FUNCTION_BLOCK Test_AssertEquals_BOOL EXTENDS TUnitTestBase
VAR
    AssertionUnderTest : TAssertion(AssertionListenerMock);
    AssertionListenerMock : TAssertionListenerMock;
    BOOL_Variable : BOOL := FALSE;
END_VAR

AssertionListenerMock.AssertionFailed  := FALSE;
AssertionListenerMock.AssertionMessage := '';
AssertionListenerMock.ExpectedAsString := '';
AssertionListenerMock.ActualAsString   := '';

// Test the assertion...
AssertionUnderTest.AssertEquals_BOOL(
    Expected := TRUE,
    Actual   := BOOL_Variable,
    VariableName := 'BOOL_Variable');
    
// Check the assertion worked...    
Assertion.AssertEquals_BOOL(
    Expected := TRUE,
    Actual   := AssertionListenerMock.AssertionFailed,
    VariableName := 'AssertionListenerMock.AssertionFailed');

// Check the assertion messages...    
Assertion.AssertEquals_STRING(
    Expected := 'AssertEquals_BOOL failed in AssertionTest: Value "BOOL_Variable"',
    Actual   := AssertionListenerMock.AssertionMessage,
    VariableName := 'AssertionListenerMock.AssertionMessage');

Assertion.AssertEquals_STRING(
    Expected := '  Expected = TRUE',
    Actual   := AssertionListenerMock.ExpectedAsString,
    VariableName := 'AssertionListenerMock.ExpectedAsString');

Assertion.AssertEquals_STRING(
    Expected := '  Actual   = FALSE',
    Actual   := AssertionListenerMock.ActualAsString,
    VariableName := 'AssertionListenerMock.ActualAsString');

TestFinished();

END_FUNCTION_BLOCK

(* stored: Version 1.1.0.1, ProductVersion 3.1.4024.4
   POU Test_AssertEquals_BOOL: Id {34d772b2-c363-42f4-9ff1-8c8ddcc83ce2}, SpecialFunc None *)
